INTERFACE itfState

METHOD mIrun : BOOL
VAR_INPUT
END_VAR
END_METHOD

END_INTERFACE

(* stored: Version 1.1.0.1, ProductVersion 3.1.4024.12
   Itf itfState: Id {3054d783-1d82-43fb-9501-0cc705668aab}
   Method mIrun: Id {b4a704ac-c5b2-46ad-90de-5b8530b3961a} *)
